// TIA Portal V20 export
// export: Created 2026-10-03T18:54:34.3273041Z, ExportSetting WithDefaults, DisplayName Totally Integrated Automation Portal, DisplayVersion V20 Update 4, DisplayName TIA Portal Openness, DisplayVersion V20 Update 4, DisplayName TIA Portal Version Control Interface, DisplayVersion V20 Update 4, DisplayName SINAMICS Startdrive Advanced, DisplayVersion V20 SP1 Update 1, DisplayName SINAMICS Startdrive G110M, G120, G120C, G120D, G120P, G115D, DisplayVersion V20 SP1 Update 1, DisplayName SINAMICS Startdrive G130, G150, S120, S150, SINAMICS MV, G220, S200, S210, DisplayVersion V20 SP1 Update 1, DisplayName STEP 7 Professional, DisplayVersion V20 Update 4, DisplayName STEP 7 Safety, DisplayVersion V20 Update 2, DisplayName WinCC Basic/Comfort/Advanced, DisplayVersion V20 Update 4, DisplayName WinCC Unified, DisplayVersion V20 Update 4
FUNCTION "SLC_WORD_READ" : Int   // FC14, SCL
TITLE = Read a whole word of a bit file
{ S7_Optimized_Access := 'TRUE' }
VERSION : 0.1
// Reads B<File>:<Element> as a number, for SLC logic that used a whole word of a bit file (MOV B3:16 N7:0,
//  EQU B3:5 0, ...). The 16 bits are named members of the DB, laid out so the word reads exactly as in the SLC.
// stored: AutoNumber true, IsIECCheckEnabled false, SetENOAutomatically false, UDAEnableTagReadback false
   VAR_INPUT
      File : DInt;   // Bit file number (3 for B3)
      Element : DInt;   // Word number (16 for B3:16)
   END_VAR
BEGIN
   // 16#84 is the DB memory area; each word is 2 bytes.
   #SLC_WORD_READ := WORD_TO_INT(PEEK_WORD(area := 16#84, dbNumber := #File, byteOffset := #Element * 2));
END_FUNCTION
